{attribute 'qualified_only'}
{attribute 'strict'}
TYPE ST100_Laser_e :
(
    RESET := 0,               // Reset
    INIT := 100,              // Initialisieren 
    READY := 999,             // READY to Start, Init Done 
    START := 1000,            // Start Zyklisch
    MOVER_FREE_OP,            // Ab here, operation without mover can be done
    waitOnMover,              // wait until the mover is there
    MOVER_NEEDED_OP,          // Ab here, a mover in position is needed to perform the action
    proceedOperation_1,       // proceed to some operation
    move_mover_to_next_piece, // move the mover to the next piece if needed
    proceedOperation_2,       // proceed to some operation
    SYNC_MOVER_LEAVE,         // MoverMan need to take the mover
    DONE := 8000,             // Ablauf beendet 
    ERROR := 9000,            // Fehler 
    _max
);
END_TYPE

(* stored: Version 1.1.0.1, ProductVersion 3.1.4024.6
   EnumerationTextList ST100_Laser_e: Id {72aa7377-c8a6-41b7-922a-e0cc3016764b} *)
